// TIA Portal project "Cau2" (V16)

(* hardware
DEVICE "S7-1200 station_1"  S7-1200 Station
   slot 0: "Rack_0"  S7-1200 Rack  Rack  V1.0
   slot 1: "PLC_1"  CPU 1214C AC/DC/Rly  6ES7 214-1BG40-0XB0  V4.2
*)

// ===== PLC "PLC_1"  CPU 1214C AC/DC/Rly =====

VAR_GLOBAL   // PLC tag table "Default tag table"
   "Start" AT %I1.1 : Bool;
   "f1" AT %M0.0 : Bool;
   "Stop" AT %I1.2 : Bool;
   "M0" AT %Q0.6 : Bool;
   "M3" AT %Q0.7 : Bool;
   "f2" AT %M0.2 : Bool;
   "T1_Off" AT %M0.1 : Bool;
   "M4" AT %Q1.1 : Bool;
   "T2_Off" AT %M0.3 : Bool;
   "f3" AT %M0.4 : Bool;
END_VAR

// folder: System blocks/Program resources

DATA_BLOCK "T1"   // DB1
{ S7_Optimized_Access := 'TRUE' }
AUTHOR : Simatic
FAMILY : IEC
NAME : IEC_TMR
VERSION : 1.0
// stored: InstanceOfName IEC_TIMER
"IEC_TIMER"
BEGIN
END_DATA_BLOCK

DATA_BLOCK "T2"   // DB2
{ S7_Optimized_Access := 'TRUE' }
AUTHOR : Simatic
FAMILY : IEC
NAME : IEC_TMR
VERSION : 1.0
// stored: InstanceOfName IEC_TIMER
"IEC_TIMER"
BEGIN
END_DATA_BLOCK

// folder: (top level)

ORGANIZATION_BLOCK "Main"   // OB1, LAD, ProgramCycle
TITLE = "Main Program Sweep (Cycle)"
{ S7_Optimized_Access := 'TRUE' }
VERSION : 0.1
   VAR_INPUT
      Initial_Call : Bool;   // Initial call of this OB
      Remanence : Bool;   // =True, if remanent data are available
   END_VAR
   VAR_TEMP   // added for the SCL form of the ladder/FBD networks
      _w1 : Bool;
   END_VAR
BEGIN

REGION Network 1
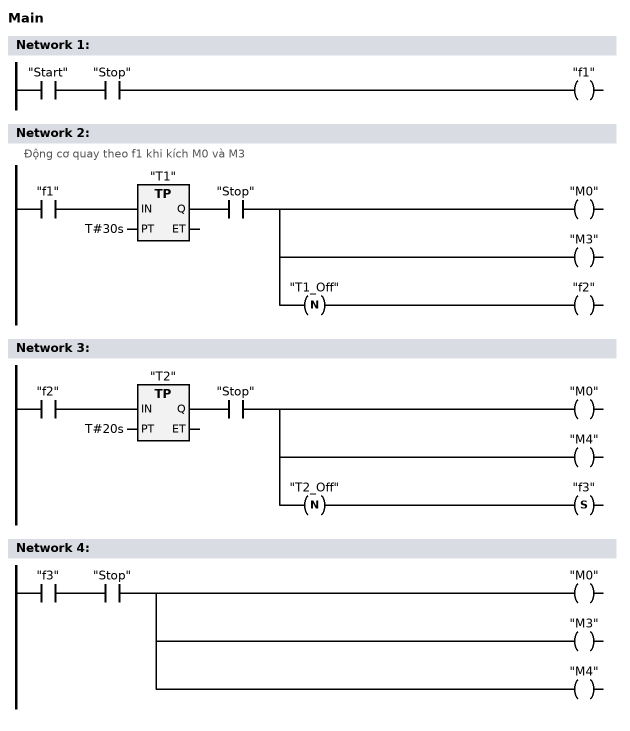
   RUNG wire#powerrail
      Contact( "Start" )
      Contact( "Stop" )
      Coil( "f1" )
   END_RUNG
   // the same network as SCL:
   "f1" := "Start" AND "Stop";
END_REGION

REGION Network 2
   // Động cơ quay theo f1 khi kích M0 và M3
   "T1".TP(IN := "f1", PT := T#30s);
   "M0" := "T1".Q AND "Stop";
   "M3" := "M0";
   #_w1 := NOT "M0" AND "T1_Off";   // falling edge
   "T1_Off" := "M0";
   "f2" := #_w1;
END_REGION

REGION Network 3
   "T2".TP(IN := "f2", PT := T#20s);
   "M0" := "T2".Q AND "Stop";
   "M4" := "M0";
   #_w1 := NOT "M0" AND "T2_Off";   // falling edge
   "T2_Off" := "M0";
   IF #_w1 THEN "f3" := TRUE; END_IF;
END_REGION

REGION Network 4
   RUNG wire#powerrail
      Contact( "f3" )
      Contact( "Stop" )
      wire#w1
      Coil( "M0" )
   END_RUNG
   RUNG wire#w1
      Coil( "M3" )
   END_RUNG
   RUNG wire#w1
      Coil( "M4" )
   END_RUNG
   // the same network as SCL:
   "M0" := "f3" AND "Stop";
   "M3" := "M0";
   "M4" := "M0";
END_REGION
END_ORGANIZATION_BLOCK